// TIA Portal V20 export
// export: Created 2026-10-03T18:54:34.8898874Z, ExportSetting WithDefaults, DisplayName Totally Integrated Automation Portal, DisplayVersion V20 Update 4, DisplayName TIA Portal Openness, DisplayVersion V20 Update 4, DisplayName TIA Portal Version Control Interface, DisplayVersion V20 Update 4, DisplayName SINAMICS Startdrive Advanced, DisplayVersion V20 SP1 Update 1, DisplayName SINAMICS Startdrive G110M, G120, G120C, G120D, G120P, G115D, DisplayVersion V20 SP1 Update 1, DisplayName SINAMICS Startdrive G130, G150, S120, S150, SINAMICS MV, G220, S200, S210, DisplayVersion V20 SP1 Update 1, DisplayName STEP 7 Professional, DisplayVersion V20 Update 4, DisplayName STEP 7 Safety, DisplayVersion V20 Update 2, DisplayName WinCC Basic/Comfort/Advanced, DisplayVersion V20 Update 4, DisplayName WinCC Unified, DisplayVersion V20 Update 4
FUNCTION "SLC_SCP" : Real   // FC25, SCL
TITLE = SLC SCP (scale with parameters)
{ S7_Optimized_Access := 'TRUE' }
VERSION : 0.1
// Replaces the SLC SCP instruction: linear scaling of Value from InMin..InMax to ScaledMin..ScaledMax.
//  Like the SLC, it extrapolates outside the input range rather than clamping.
// stored: AutoNumber true, IsIECCheckEnabled false, SetENOAutomatically false, UDAEnableTagReadback false
   VAR_INPUT
      Value : Real;   // Value to scale
      InMin : Real;   // Input value that maps to ScaledMin
      InMax : Real;   // Input value that maps to ScaledMax
      ScaledMin : Real;   // Output at InMin
      ScaledMax : Real;   // Output at InMax
   END_VAR
BEGIN
   IF #InMax = #InMin THEN
       // The SLC flags this as a math overflow; return the low end instead of dividing by zero.
       #SLC_SCP := #ScaledMin;
   ELSE
       #SLC_SCP := (#Value - #InMin) * (#ScaledMax - #ScaledMin) / (#InMax - #InMin) + #ScaledMin;
   END_IF;
END_FUNCTION
